TYPE "PLCtoMES_MainCheckOutProcessData_OP220"
VERSION : 0.1
   STRUCT
      "P-LineID" : String[18];
      "P-StationID" : String[18];
      "P-PalletNo" : Int;
      "P-PalletType" : Byte;
      "P-PalletStatus" : Byte;
      "P-CT_Total" : Real;
      "P-CT_Sub" : Array[1..20] of Real;
      "P-Data" : "PLCtoMES_OP_ProcessData_OP220";
      Reserve { S7_SetPoint := 'True'} : Array[1..1700] of Byte;
   END_STRUCT;

END_TYPE

